// SIMATIC STEP 7 (V5.x) project FC299_PNIODIAG_FILTER
// CPU: CPU314C-2 PN/DP
// station: P_ADR_BUS
// station: Hardware
// station: SIMATIC 314CPNDP
// station: P_ADR_BUS
// station: Konfiguration
// program: S7-Programm(1) - V1.8x
27.11.2012

SYMBOL_TABLE
"InstanzDB PNIODiag"	DB 126	FB 126
"DIAG_Profibus"	DB 299	DB 299	// Daten für Profibus - DP und Profinet - IO Diagnose
"DIAG_Profinet"	DB 300	DB 300
"PNIODiag"	FB 126	FB 126	// Profibus/DP und Profinet/IO-Diagnose
"DIAG_FILTER"	FC 299	FC 299	// Stationsstatus aus PNDIAG Datenbereich Filtern, DP und PN
"M20.0"	M 20.0	BOOL	// ReTrigger PUT
"M20.1"	M 20.1	BOOL	// Retrigger GET
"CYCL_EXC"	OB 1	OB 1	// Cycle Execution
"I/O_FLT1"	OB 82	OB 82	// I/O Point Fault 1
"I/O_FLT2"	OB 83	OB 83	// I/O Point Fault 2
"RACK_FLT"	OB 86	OB 86	// Loss of Rack Fault
"COMPLETE RESTART"	OB 100	OB 100	// Complete Restart
"COUNT"	SFB 47	SFB 47	// Common counter module
"RDREC"	SFB 52	SFB 52	// Read a Process Data Record
"RALRM"	SFB 54	SFB 54	// Receive Alarm Data
"BLKMOV"	SFC 20	SFC 20	// Copy Variables
"TEST_DB"	SFC 24	SFC 24	// Test Data Block
"RDSYSST"	SFC 51	SFC 51	// Read a System Status List or Partial List
"WR_REC"	SFC 58	SFC 58	// Write Data Record
"RD_REC"	SFC 59	SFC 59	// Read a Data Record
"T10"	T 10	TIMER	// Sekundentakt
"T14"	T 14	TIMER	// Watchdog GET
"T15"	T 15	TIMER	// Watchdog PUT
"DIAG_Type"	UDT 299	UDT 299	// Datentype für gefilterte Diagnose DIAG_DATA / datatype filtered diagnostic info
END_SYMBOL_TABLE

TYPE "DIAG_Type"	// UDT 299
AUTHOR : IBNS
FAMILY : Diagnose
NAME : DPDiag
VERSION : 1.8
  STRUCT
   SUM_SLAVES_DIAG : INT ;	//amount of effected slaves / Anzahl betroffene Slaves (ausgefallen oder gestört)
   LIST_SLAVES_NOT_PRESENT : ARRAY  [1 .. 128 ] OF //list of lost slaves / Liste der ausgefallenen Slaves
   BOOL ;
   LIST_SLAVES_ERROR : ARRAY  [1 .. 128 ] OF //list of faulty slaves / Liste der gestoerten Slaves
   BOOL ;
   LIST_SLAVES_MSG : ARRAY  [1 .. 128 ] OF //list of effected slaves / Liste der betroffenen Slaves (ausgefallen / gestört)
   BOOL ;
  END_STRUCT ;	
END_TYPE

// FB 126: know-how protected block, not included

FUNCTION "DIAG_FILTER" : VOID	// FC 299
TITLE = Stationsstatus aus PNIODIAG Datenbereich Filtern, DP und PN
//Filter Station status out of global DB from PNIODIAG function 
//reading from Siemens PNIODiag V1.82
//
//Cylcetime  on  314-2PN/DP FW3.3.6  approx. 0.8 ms
//
//Zykluszeit auf 314-2PN/DP FW3.3.6  ca. 0.8 ms
//
//
//System-Nr:
//First count the DP-Mastersystems, then IO-Systems in order of ther number.
//Example:
//DP-Mastersystem 2 = Systemnumber 1
//DP-Mastersystem 5 = Systemnumber 2
//IO-System     101 = Systemnumber 3
//IO-System     115 = Systemnumber 4
//
//
//Ermittlung der Systemnummer: 
//In der Reihenfolge erst DP-Mastersysteme, dann die IO-Systeme.
//
//Beispiel:
//DP-Mastersystem 2 = Systemnumber 1
//DP-Mastersystem 5 = Systemnumber 2
//IO-System     101 = Systemnumber 3
//IO-System     115 = Systemnumber 4
AUTHOR : IBNS
FAMILY : DIAGNOSE
NAME : DIAG_FIL
VERSION : 1.8
VAR_INPUT
  SYSTEM_NR : INT ;	//Systemnummer, Reihenfolge PD-PN beachten / Number of system, sequence sensitive
  PNIODiag_GLOBDB : INT ;	//Nummer Global-DB des PNIODIAG / No. Global DB of PNIODIAG function (usual 200)
  DIAG_DATA : UDT 299;	//Ziel - Datenfach für gefilterter Diagnose / DATA area with filtered diagnostic
END_VAR
VAR_OUTPUT
  ErrorDB : BOOL ;	//Fehler: PNIODIAG_DB fehlt oder zu kurz /  PNIODIAG_DB missing or to short
  ErrorsSysNr : BOOL ;	//Fehler: Systemnummer nicht erlaubt /  SystemNo. not allowed [1..48]
END_VAR
VAR_TEMP
  RetValSFC : INT ;
  DB_LENGTH : WORD ;
  GLOBDBNr : WORD ;	//Gobal-DB in word-format
  WRITE_PROT : BOOL ;
  LaengeDB : INT ;	//Erforderliche Global-DB Länge / necessary length of global DB
  System_Start : INT ;	//Startadresse für Systemnummer / Start adress of system no.
  Info_PTR_NP : DWORD ;	//Pointer auf DIAG_INFO "not Present" / Pointer local area DIAG_INFO "not Pres"
  Info_PTR_ER : DWORD ;	//Pointer auf DIAG_INFO "Error" / Pointer local area DIAG_INFO "Error"
  Info_PTR_MSG : DWORD ;	//Pointer auf DIAG_INFO "MSG" / Pointer local area DIAG_INFO "MSG" (effected)
  LoopCNTR : INT ;	//Schleifenzähler
  DataType : INT ;
  DataLoop : INT ;
  DataDBNo : INT ;
  DataArea : INT ;
  DataAdress : INT ;
  P_Any_Diag : ANY ;	//Anypointer zu Diagnosedaten / anypointer target diagdata
  DIAG_INFO : UDT 299;	//Diagnoseinformation im Lokalbereich / diag information in local area
END_VAR
BEGIN
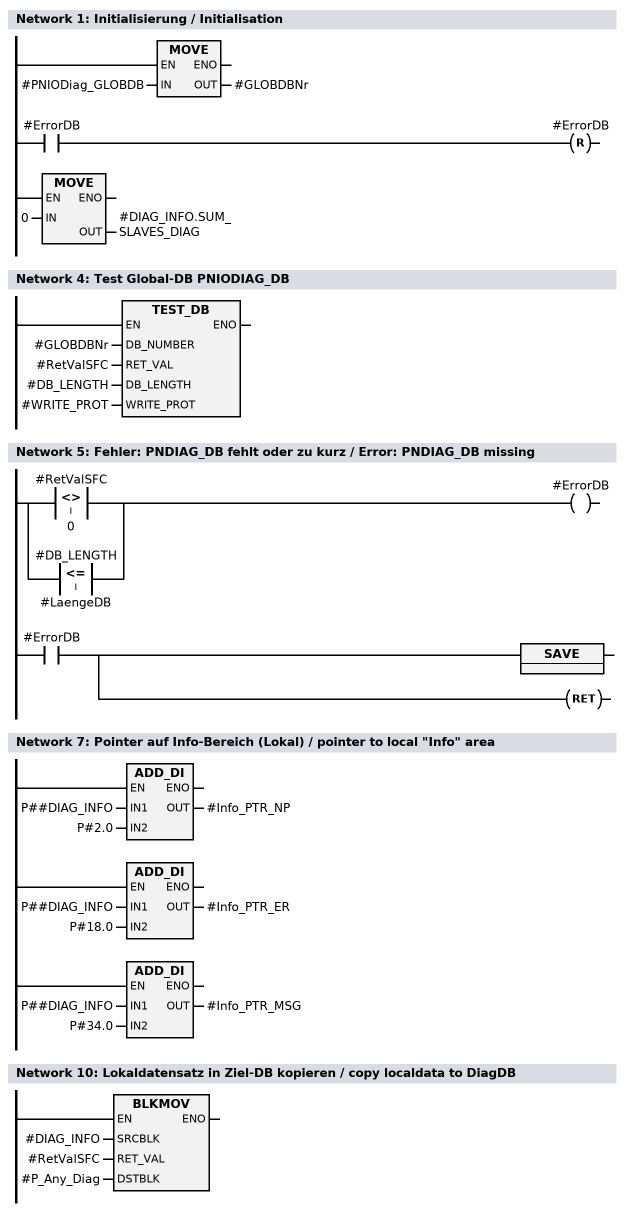
NETWORK
TITLE = Initialisierung / Initialisation
      L     #PNIODiag_GLOBDB;
      T     #GLOBDBNr;	// Global-DB Nummer in word-format
      A     #ErrorDB;
      R     #ErrorDB;	// Error-Bit reset
      L     0;
      T     #DIAG_INFO.SUM_SLAVES_DIAG;	// Slaveanzahl reset
NETWORK
TITLE = Kontrolle Systemnummer / check system number  1..48
//reserved for DP 1..32
//reserved for PN 100..115,
//all together a squence of 1..48 systems.
//
//Systemnummern für DP 1..32
//Systemnummern für PN 100..115,
//zusammen maximal 48 Systeme (DP+PN)
      L     #SYSTEM_NR;
      L     1;
      <I;
      JC    errS;	// Systemnummer kleiner 1: Fehler / system no. < 1 : Error
      TAK;
      L     48;	// Systemnummer größer 48: Fehler / system no. > 48 : Error
      <=I;
      JC    norS;
errS: S     #ErrorsSysNr;
      BEU;	// Abbruch bei falscher Systemnummer / quit if system no. is wrong
norS: R     #ErrorsSysNr;	// Reset Fehler: Systemnummer nicht erlaubt /  SystemNo. not allowed [1..48]
NETWORK
TITLE = Berechnen Min.größe Global-DB / calculating min. size Global-DB
//Minimum Size of DNDIAG_GLOBDB is depending from number of system.
//Any system needs 256 words.
//
//Die Minimalgröße des DNDIAG_GLOBDB ist abhängig von der Anzahl der Systeme.
//Jedes System belegt 256 worte im Global-DB
//
//Adresse [Byte] = (Systemnummer-1) * 256 * 2Byte + (Stationsnummer-1) * 2Byte
      L     #SYSTEM_NR;
      L     1;
      -I;
      L     256;
      *I;
      L     255;	// Max. 256 Stationen / max. 256 stations supported
      +I;
      SLW   1;
      T     #LaengeDB;	// Erforderliche Global-DB Länge / necessary length of global DB
NETWORK
TITLE = Test Global-DB PNIODIAG_DB
//PNIODIAG_DB will be generated from Siemens PNIODIAG function with PLC Startup,
//default DB200 will be generated from FB126 called in OB100
//
//Der PNIODIAG_DB wird vom Siemens PNIODIAG FC im SPS-ANlauf erzeugt,
//üblicherweise wird im OB100  der DB200 vom FB126 erzeugt.
      CALL  "TEST_DB" (
           DB_NUMBER                := #GLOBDBNr,
           RET_VAL                  := #RetValSFC,
           DB_LENGTH                := #DB_LENGTH,
           WRITE_PROT               := #WRITE_PROT);
      NOP   0;
NETWORK
TITLE = Fehler: PNDIAG_DB fehlt oder zu kurz / Error: PNDIAG_DB missing 
//Quit if PNDIAG_DB DB-Error
//
//Abbruch wenn PNDIAG_DB DB - Fehler
      A(;
      O(;
      L     #RetValSFC;
      L     0;
      <>I;
      );
      O(;
      L     #DB_LENGTH;
      L     #LaengeDB;
      <=I;
      );
      );
      =     #ErrorDB;
      A     #ErrorDB;
      SAVE;
      BEC;
NETWORK
TITLE = Berechen Anfangsadresse SystemNr. / calculation systemno. start
//Every System needs 256 word = 512 byte inside Global-DB
//
//Jedes System belegt 256 Worte = 512 bytes im Global-DB
//
//
//Adresse [Byte] = (Systemnummer-1) * 256 * 2Byte + (Stationsnummer-1) * 2Byte
      L     #SYSTEM_NR;
      L     1;
      -I;
      L     512;
      *I;
      T     #System_Start;	// Startadresse für Systemnummer / Start adress of system no.
NETWORK
TITLE = Pointer auf Info-Bereich (Lokal) / pointer to local "Info" area
      L     P##DIAG_INFO;
      L     P#2.0;
      +D;
      T     #Info_PTR_NP;	// Pointer Array "LIST_SLAVES_NOT_PRESENT"
      L     P##DIAG_INFO;
      L     P#18.0;
      +D;
      T     #Info_PTR_ER;	// Pointer Array "LIST_SLAVES_ERROR"
      L     P##DIAG_INFO;
      L     P#34.0;
      +D;
      T     #Info_PTR_MSG;	// Pointer Array "LIST_SLAVES_MSG"
NETWORK
TITLE = Teilnehmer 1..128 auswerten / Slaves 1..128 testing  => 0-127
//Adresse [Byte] = (Systemnummer-1) * 256 * 2Byte + (Stationsnummer-1) * 2Byte
//               = System_Start                   + LoopCNTR * 2
//
//Bit 0 OK
//Bit 1 Maintenance
//Bit 2 Gestört
//Bit 3 Ausgefallen
//Bit 4 Deaktiviert gewesen
//Bit 5 DPV1
//Bit 6 Maintenance gewesen
//Bit 7 Gestört gewesen
//Bit 8 Ausgefallen gewesen
//Bit 9 Deaktiviert
//Bit 10 bis 15 reserviert
      OPN   DB [#GLOBDBNr];	// Global-DB von PNIODIAG öffnen / open global DB of PNIODIAG
      L     0;
      T     #LoopCNTR;	// Teilnehmer 1 = Bit 0  / Slave 1 is bit 0
nxtT: L     #LoopCNTR;	// Teilnehmer in Zälschleife überprüfen / check slaves in loop
      SLW   1;	// LoopCNTR * 2
      L     #System_Start;
      +I;
      SLW   3;	// Pointerformat
      LAR1;
      SET;
      R     L [#Info_PTR_MSG];	// Init Ausfall oder Störung / nor present or error
      A     DBX [AR1,P#1.3];	// Ausgefallen / not present
      =     L [#Info_PTR_NP];	// Bit setzen "Teilnehmer ausgefallen" / indicate bit "not present"
      S     L [#Info_PTR_MSG];	// Ausfall oder Störung / nor present or error
      A     DBX [AR1,P#1.1];	// Maintenance   oder / or
      A     DBX [AR1,P#1.2];	// gestört / error
      =     L [#Info_PTR_ER];	// Bit setzen "Teilnehmer gestört" / indicate bit "error"
      S     L [#Info_PTR_MSG];	// Ausfall oder Störung / nor present or error
      AN    L [#Info_PTR_MSG];
      JC    kZae;	// wenn keine Störung, nicht Zählen / if no fault, do not count
      L     #DIAG_INFO.SUM_SLAVES_DIAG;
      L     1;
      +I;
      T     #DIAG_INFO.SUM_SLAVES_DIAG;	// Summenzähler erhöhen / increase sum
kZae: NOP   0;
      L     #Info_PTR_NP;	// ausgefallen / lost
      L     P#0.1;
      +D;
      T     #Info_PTR_NP;	// Zeiger auf nächstes Bit im Info-Bereich / pointer to next bit in info - area
      L     #Info_PTR_ER;	// gestört / error
      L     P#0.1;
      +D;
      T     #Info_PTR_ER;	// Zeiger auf nächstes Bit im Info-Bereich / pointer to next bit in info - area
      L     #Info_PTR_MSG;	// betroffen / effected
      L     P#0.1;
      +D;
      T     #Info_PTR_MSG;	// Zeiger auf nächstes Bit im Info-Bereich / pointer to next bit in info - area
      L     #LoopCNTR;	// Zeiger auf nächsten Teilnehmer im Global-DB / pointer to next slave in global - DB
      L     1;
      +I;
      T     #LoopCNTR;
      L     128;	// wenn alle 128 Teilnehmer bearbeitet, Schleife ende / If all 128 slaves are testet, finish loop
      <I;
      JC    nxtT;
NETWORK
TITLE = ANY für DIAGdaten bauen / create ANY for diagdata
//The parameter "DIAG_DB" for diag - DB (target) is not a pointer but an UDT.
//Therefore it is necessary to copy the missing values for "type" and "loop".
//
//Der Parameter "DIAG_DB" für den Diagnose - Ziel DB wird nicht als Pointer 
//sondern als UDT übergeben, um die Parametrierung einfacher zu gestalten.
//Daher müssen die fehlenden Argumente "Ddatentype" und "Wiederholfaktor" hinzu 
//kopiert werden.
      L     P##DIAG_DATA;	// UDT für Diagnosedaten / UDT dataset diagdata
      LAR1;
      L     W [AR1,P#0.0];
      T     #DataDBNo;
      L     W [AR1,P#2.0];
      T     #DataArea;
      L     W [AR1,P#4.0];
      T     #DataAdress;
      L     W#16#1002;	// UDT enthält keinen Typ und Wiederholfaktor / UDT does not have type and loop
      T     #DataType;	// datatype = BYTE, 10h = S7
      L     50;	// Diagnosedatenfach hat 50 byte / length of data 50 byte
      T     #DataLoop;
      L     P##P_Any_Diag;	// Anypointer zu Diagnosedaten / anypointer target diagdata
      LAR1;
      L     #DataType;
      T     LW [AR1,P#0.0];
      L     #DataLoop;
      T     LW [AR1,P#2.0];
      L     #DataDBNo;
      T     LW [AR1,P#4.0];
      L     #DataArea;
      T     LW [AR1,P#6.0];
      L     #DataAdress;
      T     LW [AR1,P#8.0];
NETWORK
TITLE = Lokaldatensatz in Ziel-DB kopieren / copy localdata to DiagDB
      CALL  "BLKMOV" (
           SRCBLK                   := #DIAG_INFO,
           RET_VAL                  := #RetValSFC,
           DSTBLK                   := #P_Any_Diag);
      NOP   0;
NETWORK
TITLE = Baustein Ende / block end
END_FUNCTION

DATA_BLOCK "InstanzDB PNIODiag"	// DB 126
AUTHOR : ICom
FAMILY : DIAGNOSE
VERSION : 0.0
"PNIODiag"
BEGIN
END_DATA_BLOCK

DATA_BLOCK "DIAG_Profibus"	// DB 299
VERSION : 0.1
  STRUCT
   D : UDT 299;
  END_STRUCT ;	
BEGIN
END_DATA_BLOCK

DATA_BLOCK "DIAG_Profinet"	// DB 300
VERSION : 0.1
  STRUCT
   D : UDT 299;
  END_STRUCT ;	
BEGIN
END_DATA_BLOCK

ORGANIZATION_BLOCK "CYCL_EXC"	// OB 1
TITLE = "Main Program Sweep (Cycle)"
//Die Bausteine für S7 sind allgemeingültige Anwendungsbeispiele von IBN-Service. 
//Die Bausteine sollen unseren Kunden bei der Programmierung und Projektierung 
//von SPS - Anwendungen unterstützen und Lösungsansätze aufzeigen. 
//Stand: 27.11.2012
//
//Diese sind kein kostenpflichtiges Produkt unseres Unternehmens. 
//
//Ein Anspruch auf Gewährleistung, Fehlerbeseitigung und Update besteht für den 
//Anwender nicht. 
//Ebenso schließen wir die Haftung für Schäden, die infolge des Einsatzes dieser 
//Bausteine auftreten, ausdrücklich aus.
//
//Für Rückmeldungen, Fragen und Verbesserungsvorschläge sind wir stets dankbar.
//
//IBN-Service Jürgen Müller
// Gagernstraße 17
// 57072 Siegen
//
// Tel./Fax:  0271 / 31 74 286
// Mobil   :  0171 / 17 45 330
// e-mail  :  info@ibn-service.com 
// http://www.ibn-service.com
VERSION : 0.1
VAR_TEMP
  OB1_EV_CLASS : BYTE ;	//Bits 0-3 = 1 (Coming event), Bits 4-7 = 1 (Event class 1)
  OB1_SCAN_1 : BYTE ;	//1 (Cold restart scan 1 of OB 1), 3 (Scan 2-n of OB 1)
  OB1_PRIORITY : BYTE ;	//Priority of OB Execution
  OB1_OB_NUMBR : BYTE ;	//1 (Organization block 1, OB1)
  OB1_RESERVED_1 : BYTE ;	//Reserved for system
  OB1_RESERVED_2 : BYTE ;	//Reserved for system
  OB1_PREV_CYCLE : INT ;	//Cycle time of previous OB1 scan (milliseconds)
  OB1_MIN_CYCLE : INT ;	//Minimum cycle time of OB1 (milliseconds)
  OB1_MAX_CYCLE : INT ;	//Maximum cycle time of OB1 (milliseconds)
  OB1_DATE_TIME : DATE_AND_TIME ;	//Date and time OB1 started
END_VAR
BEGIN
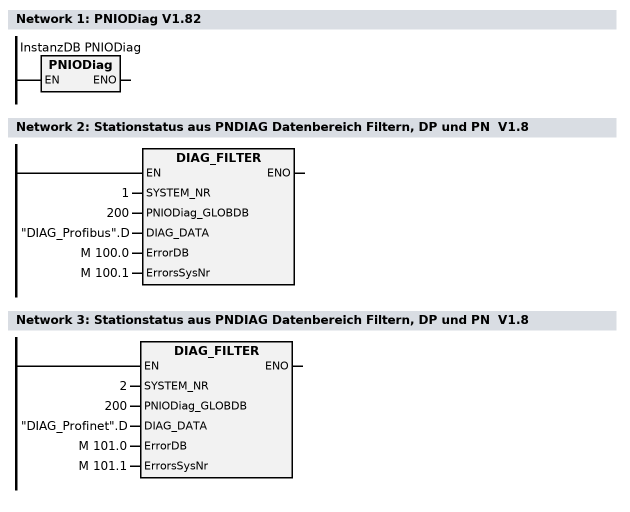
NETWORK
TITLE = PNIODiag V1.82
//IN0:  Datenbausteinnummer Diagnosedaten
//OUT1: Status-Wort
      CALL  "PNIODiag" , "InstanzDB PNIODiag";
NETWORK
TITLE = Stationstatus aus PNDIAG Datenbereich Filtern, DP und PN  V1.8
//System Nr. 1 = Profibus
      CALL  "DIAG_FILTER" (
           SYSTEM_NR                := 1,
           PNIODiag_GLOBDB          := 200,
           DIAG_DATA                := "DIAG_Profibus".D,
           ErrorDB                  := M 100.0,
           ErrorsSysNr              := M 100.1);
      NOP   0;
NETWORK
TITLE = Stationstatus aus PNDIAG Datenbereich Filtern, DP und PN  V1.8
//System Nr. 2 = Profinet
      CALL  "DIAG_FILTER" (
           SYSTEM_NR                := 2,
           PNIODiag_GLOBDB          := 200,
           DIAG_DATA                := "DIAG_Profinet".D,
           ErrorDB                  := M 101.0,
           ErrorsSysNr              := M 101.1);
      NOP   0;
NETWORK
TITLE = Baustein Ende
END_ORGANIZATION_BLOCK

ORGANIZATION_BLOCK "I/O_FLT1"	// OB 82
TITLE = "I/O Point Fault"
VERSION : 0.1
VAR_TEMP
  OB82_EV_CLASS : BYTE ;	//16#39, Event class 3, Entering event state, Internal fault event
  OB82_FLT_ID : BYTE ;	//16#XX, Fault identifcation code
  OB82_PRIORITY : BYTE ;	//Priority of OB Execution
  OB82_OB_NUMBR : BYTE ;	//82 (Organization block 82, OB82)
  OB82_RESERVED_1 : BYTE ;	//Reserved for system
  OB82_IO_FLAG : BYTE ;	//Input (01010100), Output (01010101)
  OB82_MDL_ADDR : WORD ;	//Base address of module with fault
  OB82_MDL_DEFECT : BOOL ;	//Module defective
  OB82_INT_FAULT : BOOL ;	//Internal fault
  OB82_EXT_FAULT : BOOL ;	//External fault
  OB82_PNT_INFO : BOOL ;	//Point information
  OB82_EXT_VOLTAGE : BOOL ;	//External voltage low
  OB82_FLD_CONNCTR : BOOL ;	//Field wiring connector missing
  OB82_NO_CONFIG : BOOL ;	//Module has no configuration data
  OB82_CONFIG_ERR : BOOL ;	//Module has configuration error
  OB82_MDL_TYPE : BYTE ;	//Type of module
  OB82_SUB_MDL_ERR : BOOL ;	//Sub-Module is missing or has error
  OB82_COMM_FAULT : BOOL ;	//Communication fault
  OB82_MDL_STOP : BOOL ;	//Module is stopped
  OB82_WTCH_DOG_FLT : BOOL ;	//Watch dog timer stopped module
  OB82_INT_PS_FLT : BOOL ;	//Internal power supply fault
  OB82_PRIM_BATT_FLT : BOOL ;	//Primary battery is in fault
  OB82_BCKUP_BATT_FLT : BOOL ;	//Backup battery is in fault
  OB82_RESERVED_2 : BOOL ;	//Reserved for system
  OB82_RACK_FLT : BOOL ;	//Rack fault, only for bus interface module
  OB82_PROC_FLT : BOOL ;	//Processor fault
  OB82_EPROM_FLT : BOOL ;	//EPROM fault
  OB82_RAM_FLT : BOOL ;	//RAM fault
  OB82_ADU_FLT : BOOL ;	//ADU fault
  OB82_FUSE_FLT : BOOL ;	//Fuse fault
  OB82_HW_INTR_FLT : BOOL ;	//Hardware interupt input in fault
  OB82_RESERVED_3 : BOOL ;	//Reserved for system
  OB82_DATE_TIME : DATE_AND_TIME ;	//Date and time OB82 started
END_VAR
BEGIN
NETWORK
TITLE = PNIODiag V1.82
//IN0:  Datenbausteinnummer Diagnosedaten
//OUT1: Status-Wort
      CALL  "PNIODiag" , "InstanzDB PNIODiag";
END_ORGANIZATION_BLOCK

ORGANIZATION_BLOCK "I/O_FLT2"	// OB 83
TITLE = "I/O Point Fault"
VERSION : 0.1
VAR_TEMP
  OB83_EV_CLASS : BYTE ;	//16#38/39, Event class 3, module inserted/removed (8/9)
  OB83_FLT_ID : BYTE ;	//16#XX, Fault identifcation code
  OB83_PRIORITY : BYTE ;	//Priority of OB Execution
  OB83_OB_NUMBR : BYTE ;	//83 (Organization block 83, OB83)
  OB83_RESERVED_1 : BYTE ;	//Reserved for system
  OB83_MDL_ID : BYTE ;	//Input module (01010100), Output module (01010101)
  OB83_MDL_ADDR : WORD ;	//Base address of module with point fault
  OB83_RACK_NUM : INT ;	//Number of rack that has module with point fault
  OB83_MDL_TYPE : WORD ;	//Module type with point fault
  OB83_DATE_TIME : DATE_AND_TIME ;	//Date and time OB83 started
END_VAR
BEGIN
NETWORK
TITLE = PNIODiag V1.82
//IN0:  Datenbausteinnummer Diagnosedaten
//OUT1: Status-Wort
      CALL  "PNIODiag" , "InstanzDB PNIODiag";
END_ORGANIZATION_BLOCK

ORGANIZATION_BLOCK "RACK_FLT"	// OB 86
TITLE = "Loss Of Rack Fault"
VERSION : 0.1
VAR_TEMP
  OB86_EV_CLASS : BYTE ;	//16#38/39 Event class 3
  OB86_FLT_ID : BYTE ;	//16#C1/C4/C5, Fault identifcation code
  OB86_PRIORITY : BYTE ;	//Priority of OB Execution
  OB86_OB_NUMBR : BYTE ;	//86 (Organization block 86, OB86)
  OB86_RESERVED_1 : BYTE ;	//Reserved for system
  OB86_RESERVED_2 : BYTE ;	//Reserved for system
  OB86_MDL_ADDR : WORD ;	//Base address of IM module in rack with fault
  OB86_RACKS_FLTD : ARRAY  [0 .. 31 ] OF BOOL ;	//Racks in fault
  OB86_DATE_TIME : DATE_AND_TIME ;	//Date and time OB86 started
END_VAR
BEGIN
NETWORK
TITLE = PNIODiag V1.82
//IN0:  Datenbausteinnummer Diagnosedaten
//OUT1: Status-Wort
      CALL  "PNIODiag" , "InstanzDB PNIODiag";
END_ORGANIZATION_BLOCK

ORGANIZATION_BLOCK "COMPLETE RESTART"	// OB 100
TITLE = "Complete Restart"
VERSION : 0.1
VAR_TEMP
  OB100_EV_CLASS : BYTE ;	//16#13, Event class 1, Entering event state, Event logged in diagnostic buffer
  OB100_STRTUP : BYTE ;	//16#81/82/83/84 Method of startup
  OB100_PRIORITY : BYTE ;	//Priority of OB Execution
  OB100_OB_NUMBR : BYTE ;	//100 (Organization block 100, OB100)
  OB100_RESERVED_1 : BYTE ;	//Reserved for system
  OB100_RESERVED_2 : BYTE ;	//Reserved for system
  OB100_STOP : WORD ;	//Event that caused CPU to stop (16#4xxx)
  OB100_STRT_INFO : DWORD ;	//Information on how system started
  OB100_DATE_TIME : DATE_AND_TIME ;	//Date and time OB100 started
END_VAR
BEGIN
NETWORK
TITLE = PNIODiag V1.82
//IN0:  Datenbausteinnummer Diagnosedaten
//OUT1: Status-Wort
      CALL  "PNIODiag" , "InstanzDB PNIODiag";
END_ORGANIZATION_BLOCK
